// TIA Portal V17 export
// export: Created 2025-03-13T10:31:02.7493428Z, ExportSetting WithDefaults, DisplayName Totally Integrated Automation Portal, DisplayVersion V17 Update 8, DisplayName TIA Portal Openness, DisplayVersion V17 Update 8, DisplayName TIA Portal Version Control Interface, DisplayVersion V17, DisplayName SINAMICS Startdrive Advanced, DisplayVersion V17 SP2, DisplayName SINAMICS Startdrive G110M, G120, G120C, G120D, G120P, G115D, DisplayVersion V17 SP2, DisplayName SINAMICS Startdrive G130, G150, S120, S150, SINAMICS MV, S210, DisplayVersion V17 SP2, DisplayName STEP 7 Professional, DisplayVersion V17 Update 8, DisplayName SINUMERIK ONE STEP 7 Toolbox, DisplayVersion V17 Update 12, DisplayName SINUMERIK 840D sl STEP 7 Toolbox, DisplayVersion V17 Update 12, DisplayName STEP 7 Safety, DisplayVersion V17 Update 6, DisplayName WinCC Advanced, DisplayVersion V17 Update 8
DATA_BLOCK "DB1030_TEST_STOP"   // DB1030
{ S7_Optimized_Access := 'FALSE'; DB_Accessible_From_OPC_UA := 'FALSE' }
AUTHOR : ETXETAR
VERSION : 1.0
// stored: AutoNumber false, DBAccessibleFromOPCUA false, DBAccessibleFromWebserver true, IsOnlyStoredInLoadMemory false, IsWriteProtectedInAS false
   VAR
      TEST_STP_GEN_COND : Bool;   // TEST STOP GENERAL CONDITIONS / GENERAL CONDITIONS
      TEST_STP_INIT_COND : Bool;   // TEST STOP INITIAL CONDITIONS / INITIAL CONDITIONS
      TST_STP_FIRST_SCAN_REQUEST : Bool;   // FIRST SCAN REQUEST
      TEST_STP_START_REQ : Bool;   // TEST STOP START REQUEST / START REQUEST
      TEST_STP_CMD : Bool;   // TEST STOP COMMAND / COMMAND
      TEST_STP_CMD_P : Bool;   // TEST STOP COMMAND PULSE / COMMAND PULSE
      TEST_STP_SQ_IN_PROCESS : Bool;   // TEST STOP SEQUENCE IN PROCESS / SEQUENCE IN PROCESS
      TEST_STP_TST_BRK_AX_1 : Bool;   // TEST STOP TEST BRAKE AXIS 1 / BRAKE TEST AXIS 1
      TEST_STP_TST_BRK_AX_2 : Bool;   // TEST STOP TEST BRAKE AXIS 2 / BRAKE TEST AXIS 2
      TEST_STP_TST_BRK_AX_3 : Bool;   // TEST STOP TEST BRAKE AXIS 3 / BRAKE TEST AXIS 3
      TEST_STP_TST_BRK_AX_4 : Bool;   // TEST STOP TEST BRAKE AXIS 4 / BRAKE TEST AXIS 4
      TEST_STP_TST_BRK_AX_5 : Bool;   // TEST STOP TEST BRAKE AXIS 5 / BRAKE TEST AXIS 5
      TEST_STP_TST_BRK_AX_6 : Bool;   // TEST STOP TEST BRAKE AXIS 6 / BRAKE TEST AXIS 6
      TEST_STP_TST_BRK_AX_7 : Bool;   // TEST STOP TEST BRAKE AXIS 7 / BRAKE TEST AXIS 7
      TEST_STP_TST_BRK_AX_8 : Bool;   // TEST STOP TEST BRAKE AXIS 8 / BRAKE TEST AXIS 8
      TEST_STP_TST_BRK_AX_9 : Bool;   // TEST STOP TEST BRAKE AXIS 9 / BRAKE TEST AXIS 9
      TEST_STP_TST_BRK_AX_10 : Bool;   // TEST STOP TEST BRAKE AXIS 10 / BRAKE TEST AXIS 10
      TEST_STP_TST_BRK_AX_11 : Bool;   // TEST STOP TEST BRAKE AXIS 11 / BRAKE TEST AXIS 11
      TEST_STP_TST_BRK_AX_12 : Bool;   // TEST STOP TEST BRAKE AXIS 12 / BRAKE TEST AXIS 12
      TEST_STP_TST_BRK_AX_13 : Bool;   // TEST STOP TEST BRAKE AXIS 13 / BRAKE TEST AXIS 13
      TEST_STP_TST_BRK_AX_14 : Bool;   // TEST STOP TEST BRAKE AXIS 14 / BRAKE TEST AXIS 14
      TEST_STP_TST_BRK_AX_15 : Bool;   // TEST STOP TEST BRAKE AXIS15 / BRAKE TEST AXIS 15
      TEST_STP_TST_BRK_AX_16 : Bool;   // TEST STOP TEST BRAKE AXIS 16 / BRAKE TEST AXIS 16
      TEST_STP_TST_BRK_AX_17 : Bool;   // TEST STOP TEST BRAKE AXIS 17 / BRAKE TEST AXIS 17
      TEST_STP_TST_BRK_AX_18 : Bool;   // TEST STOP TEST BRAKE AXIS 18 / BRAKE TEST AXIS 18
      TEST_STP_TST_BRK_AX_19 : Bool;   // TEST STOP TEST BRAKE AXIS 19 / BRAKE TEST AXIS 19
      TEST_STP_TST_BRK_AX_20 : Bool;   // TEST STOP TEST BRAKE AXIS 20 / BRAKE TEST AXIS 20
      TEST_STP_TST_BRK_AX_21 : Bool;   // TEST STOP TEST BRAKE AXIS 21 / BRAKE TEST AXIS 21
      TEST_STP_TST_BRK_AX_22 : Bool;   // TEST STOP TEST BRAKE AXIS 22 / BRAKE TEST AXIS 22
      TEST_STP_TST_BRK_AX_23 : Bool;   // TEST STOP TEST BRAKE AXIS 23 / BRAKE TEST AXIS 23
      TEST_STP_TST_BRK_AX_24 : Bool;   // TEST STOP TEST BRAKE AXIS 24 / BRAKE TEST AXIS 24
      TEST_STP_TST_BRK_AX_25 : Bool;   // TEST STOP TEST BRAKE AXIS 25 / BRAKE TEST AXIS 25
      TEST_STP_TST_BRK_AX_26 : Bool;   // TEST STOP TEST BRAKE AXIS 26 / BRAKE TEST AXIS 26
      TEST_STP_TST_BRK_AX_27 : Bool;   // TEST STOP TEST BRAKE AXIS 27 / BRAKE TEST AXIS 27
      TEST_STP_TST_BRK_AX_28 : Bool;   // TEST STOP TEST BRAKE AXIS 28 / BRAKE TEST AXIS 28
      TEST_STP_TST_BRK_AX_29 : Bool;   // TEST STOP TEST BRAKE AXIS 29 / BRAKE TEST AXIS 29
      TEST_STP_TST_BRK_AX_30 : Bool;   // TEST STOP TEST BRAKE AXIS 30 / BRAKE TEST AXIS 30
      TEST_STP_TST_BRK_AX_31 : Bool;   // TEST STOP TEST BRAKE AXIS 31 / BRAKE TEST AXIS 31
      TEST_STP_TST_BRK_AX_32 : Bool;   // TEST STOP TEST BRAKE AXIS 32 / BRAKE TEST AXIS 32
      TEST_STP_TST_BRK_AX_33 : Bool;   // TEST STOP TEST BRAKE AXIS 33 / BRAKE TEST AXIS 33
      TEST_STP_TST_BRK_AX_34 : Bool;   // TEST STOP TEST BRAKE AXIS 34 / BRAKE TEST AXIS 34
      TEST_STP_TST_BRK_AX_35 : Bool;   // TEST STOP TEST BRAKE AXIS 35 / BRAKE TEST AXIS 35
      TEST_STP_TST_BRK_AX_36 : Bool;   // TEST STOP TEST BRAKE AXIS 36 / BRAKE TEST AXIS 36
      TEST_STP_TST_BRK_AX_37 : Bool;   // TEST STOP TEST BRAKE AXIS 37 / BRAKE TEST AXIS 37
      TEST_STP_TST_BRK_AX_38 : Bool;   // TEST STOP TEST BRAKE AXIS 38 / BRAKE TEST AXIS 38
      TEST_STP_TST_BRK_DONE : Bool;   // TEST STOP TEST BRAKE AXIS 39 / BRAKE TEST DONE
      TEST_STP_INT_P_REQ : Bool;   // TEST STOP START INTERNAL PULSES REQUEST / INTERNAL PULSES REQUEST
      TEST_STP_INT_P_REQ_AUX : Bool;   // TEST STOP START INTERNAL PULSES REQUEST PULSE / INTERNAL PULSES REQUEST AUXILIARY
      TEST_STP_INT_P_DONE : Bool;   // TEST STOP START INTERNAL PULSES DONE / INTERNAL PULSES DONE
      TEST_STP_INT_P_ANY_AX_REQ : Bool;   // TEST STOP START INTERNAL PULSES ANY AXIS REQUEST / INTERNAL PULSES ANY AXIS REQUEST
      TEST_STP_RST_PLC_CNC_SEQ : Bool;   // TEST STOP RESET PLC AND CNC / RESET PLC CNC SEQUENCE
      TEST_STP_DONE_LOCKED : Bool;   // TEST STOP DONE LOCKED / DONE LOCKED
      TEST_STP_8_HOURS : Bool;   // TEST STOP DONE LOCKED / 8 HOURS
      TEST_STP_SQ_DONE : Bool;   // TEST STOP SEQUENCE DONE / SEQUENCE DONE
      TEST_STP_SQ_TIME_EXCEEDED : Bool;   // TEST STOP SEQUENCE TIME EXCEEDED / SEQUENCE TIME EXCEEDED
      TEST_STP_FDBCK_OVERTIME : Bool;   // TEST STOP FEEDBACK TIME EXCEEDED / FEEDBACK OVERTIME
      TEST_STP_INTERNAL_P_F_AX_1 : Bool;   // TEST STOP START INTERNAL PULSES FAULT AXIS 1 / INTERNAL PULSES FAULT AXIS 1
      TEST_STP_INTERNAL_P_F_AX_2 : Bool;   // TEST STOP START INTERNAL PULSES FAULT AXIS 2 / INTERNAL PULSES FAULT AXIS 2
      TEST_STP_INTERNAL_P_F_AX_3 : Bool;   // TEST STOP START INTERNAL PULSES FAULT AXIS 3 / INTERNAL PULSES FAULT AXIS 3
      TEST_STP_INTERNAL_P_F_AX_4 : Bool;   // TEST STOP START INTERNAL PULSES FAULT AXIS 4 / INTERNAL PULSES FAULT AXIS 4
      TEST_STP_INTERNAL_P_F_AX_5 : Bool;   // TEST STOP START INTERNAL PULSES FAULT AXIS 5 / INTERNAL PULSES FAULT AXIS 5
      TEST_STP_INTERNAL_P_F_AX_6 : Bool;   // TEST STOP START INTERNAL PULSES FAULT AXIS 6 / INTERNAL PULSES FAULT AXIS 6
      TEST_STP_INTERNAL_P_F_AX_7 : Bool;   // TEST STOP START INTERNAL PULSES FAULT AXIS 7 / INTERNAL PULSES FAULT AXIS 7
      TEST_STP_INTERNAL_P_F_AX_8 : Bool;   // TEST STOP START INTERNAL PULSES FAULT AXIS 8 / INTERNAL PULSES FAULT AXIS 8
      TEST_STP_INTERNAL_P_F_AX_9 : Bool;   // TEST STOP START INTERNAL PULSES FAULT AXIS 9 / INTERNAL PULSES FAULT AXIS 9
      TEST_STP_INTERNAL_P_F_AX_10 : Bool;   // TEST STOP START INTERNAL PULSES FAULT AXIS 10 / INTERNAL PULSES FAULT AXIS 10
      TEST_STP_INTERNAL_P_F_AX_11 : Bool;   // TEST STOP START INTERNAL PULSES FAULT AXIS 11 / INTERNAL PULSES FAULT AXIS 11
      TEST_STP_INTERNAL_P_F_AX_12 : Bool;   // TEST STOP START INTERNAL PULSES FAULT AXIS 12 / INTERNAL PULSES FAULT AXIS 12
      TEST_STP_INTERNAL_P_F_AX_13 : Bool;   // TEST STOP START INTERNAL PULSES FAULT AXIS 13 / INTERNAL PULSES FAULT AXIS 13
      TEST_STP_INTERNAL_P_F_AX_14 : Bool;   // TEST STOP START INTERNAL PULSES FAULT AXIS 14 / INTERNAL PULSES FAULT AXIS 14
      TEST_STP_INTERNAL_P_F_AX_15 : Bool;   // TEST STOP START INTERNAL PULSES FAULT AXIS 15 / INTERNAL PULSES FAULT AXIS 15
      TEST_STP_INTERNAL_P_F_AX_16 : Bool;   // TEST STOP START INTERNAL PULSES FAULT AXIS 16 / INTERNAL PULSES FAULT AXIS 16
      TEST_STP_INTERNAL_P_F_AX_17 : Bool;   // TEST STOP START INTERNAL PULSES FAULT AXIS 17 / INTERNAL PULSES FAULT AXIS 17
      TEST_STP_INTERNAL_P_F_AX_18 : Bool;   // TEST STOP START INTERNAL PULSES FAULT AXIS 18 / INTERNAL PULSES FAULT AXIS 18
      TEST_STP_INTERNAL_P_F_AX_19 : Bool;   // TEST STOP START INTERNAL PULSES FAULT AXIS 19 / INTERNAL PULSES FAULT AXIS 19
      TEST_STP_INTERNAL_P_F_AX_20 : Bool;   // TEST STOP START INTERNAL PULSES FAULT AXIS 20 / INTERNAL PULSES FAULT AXIS 20
      TEST_STP_INTERNAL_P_F_AX_21 : Bool;   // TEST STOP START INTERNAL PULSES FAULT AXIS 21 / INTERNAL PULSES FAULT AXIS 21
      TEST_STP_INTERNAL_P_F_AX_22 : Bool;   // TEST STOP START INTERNAL PULSES FAULT AXIS 22 / INTERNAL PULSES FAULT AXIS 22
      TEST_STP_INTERNAL_P_F_AX_23 : Bool;   // TEST STOP START INTERNAL PULSES FAULT AXIS 23 / INTERNAL PULSES FAULT AXIS 23
      TEST_STP_INTERNAL_P_F_AX_24 : Bool;   // TEST STOP START INTERNAL PULSES FAULT AXIS 24 / INTERNAL PULSES FAULT AXIS 24
      TEST_STP_INTERNAL_P_F_AX_25 : Bool;   // TEST STOP START INTERNAL PULSES FAULT AXIS 25 / INTERNAL PULSES FAULT AXIS 25
      TEST_STP_INTERNAL_P_F_AX_26 : Bool;   // TEST STOP START INTERNAL PULSES FAULT AXIS 26 / INTERNAL PULSES FAULT AXIS 26
      TEST_STP_INTERNAL_P_F_AX_27 : Bool;   // TEST STOP START INTERNAL PULSES FAULT AXIS 27 / INTERNAL PULSES FAULT AXIS 27
      TEST_STP_INTERNAL_P_F_AX_28 : Bool;   // TEST STOP START INTERNAL PULSES FAULT AXIS 28 / INTERNAL PULSES FAULT AXIS 28
      TEST_STP_INTERNAL_P_F_AX_29 : Bool;   // TEST STOP START INTERNAL PULSES FAULT AXIS 29 / INTERNAL PULSES FAULT AXIS 29
      TEST_STP_INTERNAL_P_F_AX_30 : Bool;   // TEST STOP START INTERNAL PULSES FAULT AXIS 30 / INTERNAL PULSES FAULT AXIS 30
      TEST_STP_INTERNAL_P_F_AX_31 : Bool;   // TEST STOP START INTERNAL PULSES FAULT AXIS 31 / INTERNAL PULSES FAULT AXIS 31
      TEST_STP_INTERNAL_P_F_AX_32 : Bool;   // TEST STOP START INTERNAL PULSES FAULT AXIS 32 / INTERNAL PULSES FAULT AXIS 32
      TEST_STP_INTERNAL_P_F_AX_33 : Bool;   // TEST STOP START INTERNAL PULSES FAULT AXIS 33 / INTERNAL PULSES FAULT AXIS 33
      TEST_STP_INTERNAL_P_F_AX_34 : Bool;   // TEST STOP START INTERNAL PULSES FAULT AXIS 34 / INTERNAL PULSES FAULT AXIS 34
      TEST_STP_INTERNAL_P_F_AX_35 : Bool;   // TEST STOP START INTERNAL PULSES FAULT AXIS 35 / INTERNAL PULSES FAULT AXIS 35
      TEST_STP_INTERNAL_P_F_AX_36 : Bool;   // TEST STOP START INTERNAL PULSES FAULT AXIS 36 / INTERNAL PULSES FAULT AXIS 36
      TEST_STP_INTERNAL_P_F_AX_37 : Bool;   // TEST STOP START INTERNAL PULSES FAULT AXIS 37 / INTERNAL PULSES FAULT AXIS 37
      TEST_STP_INTERNAL_P_F_AX_38 : Bool;   // TEST STOP START INTERNAL PULSES FAULT AXIS 38 / INTERNAL PULSES FAULT AXIS 38
      TEST_STP_INTERNAL_P_F_AX_39 : Bool;   // TEST STOP START INTERNAL PULSES FAULT AXIS 39 / INTERNAL PULSES FAULT AXIS 39
      TEST_STP_TST_BRK_F_AX_1 : Bool;   // TEST STOP TEST BRAKE FAULT AXIS 1 / BRAKE TEST FAULT AXIS 1
      TEST_STP_TST_BRK_F_AX_2 : Bool;   // TEST STOP TEST BRAKE FAULT AXIS 2 / BRAKE TEST FAULT AXIS 2
      TEST_STP_TST_BRK_F_AX_3 : Bool;   // TEST STOP TEST BRAKE FAULT AXIS 3 / BRAKE TEST FAULT AXIS 3
      TEST_STP_TST_BRK_F_AX_4 : Bool;   // TEST STOP TEST BRAKE FAULT AXIS 4 / BRAKE TEST FAULT AXIS 4
      TEST_STP_TST_BRK_F_AX_5 : Bool;   // TEST STOP TEST BRAKE FAULT AXIS 5 / BRAKE TEST FAULT AXIS 5
      TEST_STP_TST_BRK_F_AX_6 : Bool;   // TEST STOP TEST BRAKE FAULT AXIS 6 / BRAKE TEST FAULT AXIS 6
      TEST_STP_TST_BRK_F_AX_7 : Bool;   // TEST STOP TEST BRAKE FAULT AXIS 7 / BRAKE TEST FAULT AXIS 7
      TEST_STP_TST_BRK_F_AX_8 : Bool;   // TEST STOP TEST BRAKE FAULT AXIS 8 / BRAKE TEST FAULT AXIS 8
      TEST_STP_TST_BRK_F_AX_9 : Bool;   // TEST STOP TEST BRAKE FAULT AXIS 9 / BRAKE TEST FAULT AXIS 9
      TEST_STP_TST_BRK_F_AX_10 : Bool;   // TEST STOP TEST BRAKE FAULT AXIS 10 / BRAKE TEST FAULT AXIS 10
      TEST_STP_TST_BRK_F_AX_11 : Bool;   // TEST STOP TEST BRAKE FAULT AXIS 11 / BRAKE TEST FAULT AXIS 11
      TEST_STP_TST_BRK_F_AX_12 : Bool;   // TEST STOP TEST BRAKE FAULT AXIS 12 / BRAKE TEST FAULT AXIS 12
      TEST_STP_TST_BRK_F_AX_13 : Bool;   // TEST STOP TEST BRAKE FAULT AXIS 13 / BRAKE TEST FAULT AXIS 13
      TEST_STP_TST_BRK_F_AX_14 : Bool;   // TEST STOP TEST BRAKE FAULT AXIS 14 / BRAKE TEST FAULT AXIS 14
      TEST_STP_TST_BRK_F_AX_15 : Bool;   // TEST STOP TEST BRAKE FAULT AXIS 15 / BRAKE TEST FAULT AXIS 15
      TEST_STP_TST_BRK_F_AX_16 : Bool;   // TEST STOP TEST BRAKE FAULT AXIS 16 / BRAKE TEST FAULT AXIS 16
      TEST_STP_TST_BRK_F_AX_17 : Bool;   // TEST STOP TEST BRAKE FAULT AXIS 17 / BRAKE TEST FAULT AXIS 17
      TEST_STP_TST_BRK_F_AX_18 : Bool;   // TEST STOP TEST BRAKE FAULT AXIS 18 / BRAKE TEST FAULT AXIS 18
      TEST_STP_TST_BRK_F_AX_19 : Bool;   // TEST STOP TEST BRAKE FAULT AXIS 19 / BRAKE TEST FAULT AXIS 19
      TEST_STP_TST_BRK_F_AX_20 : Bool;   // TEST STOP TEST BRAKE FAULT AXIS 20 / BRAKE TEST FAULT AXIS 20
      TEST_STP_TST_BRK_F_AX_21 : Bool;   // TEST STOP TEST BRAKE FAULT AXIS 21 / BRAKE TEST FAULT AXIS 21
      TEST_STP_TST_BRK_F_AX_22 : Bool;   // TEST STOP TEST BRAKE FAULT AXIS 22 / BRAKE TEST FAULT AXIS 22
      TEST_STP_TST_BRK_F_AX_23 : Bool;   // TEST STOP TEST BRAKE FAULT AXIS 23 / BRAKE TEST FAULT AXIS 23
      TEST_STP_TST_BRK_F_AX_24 : Bool;   // TEST STOP TEST BRAKE FAULT AXIS 24 / BRAKE TEST FAULT AXIS 24
      TEST_STP_TST_BRK_F_AX_25 : Bool;   // TEST STOP TEST BRAKE FAULT AXIS 25 / BRAKE TEST FAULT AXIS 25
      TEST_STP_TST_BRK_F_AX_26 : Bool;   // TEST STOP TEST BRAKE FAULT AXIS 26 / BRAKE TEST FAULT AXIS 26
      TEST_STP_TST_BRK_F_AX_27 : Bool;   // TEST STOP TEST BRAKE FAULT AXIS 27 / BRAKE TEST FAULT AXIS 27
      TEST_STP_TST_BRK_F_AX_28 : Bool;   // TEST STOP TEST BRAKE FAULT AXIS 28 / BRAKE TEST FAULT AXIS 28
      TEST_STP_TST_BRK_F_AX_29 : Bool;   // TEST STOP TEST BRAKE FAULT AXIS 29 / BRAKE TEST FAULT AXIS 29
      TEST_STP_TST_BRK_F_AX_30 : Bool;   // TEST STOP TEST BRAKE FAULT AXIS 30 / BRAKE TEST FAULT AXIS 30
      TEST_STP_TST_BRK_F_AX_31 : Bool;   // TEST STOP TEST BRAKE FAULT AXIS 31 / BRAKE TEST FAULT AXIS 31
      TEST_STP_TST_BRK_F_AX_32 : Bool;   // TEST STOP TEST BRAKE FAULT AXIS 32 / BRAKE TEST FAULT AXIS 32
      TEST_STP_TST_BRK_F_AX_33 : Bool;   // TEST STOP TEST BRAKE FAULT AXIS 33 / BRAKE TEST FAULT AXIS 33
      TEST_STP_TST_BRK_F_AX_34 : Bool;   // TEST STOP TEST BRAKE FAULT AXIS 34 / BRAKE TEST FAULT AXIS 34
      TEST_STP_TST_BRK_F_AX_35 : Bool;   // TEST STOP TEST BRAKE FAULT AXIS 35 / BRAKE TEST FAULT AXIS 35
      TEST_STP_TST_BRK_F_AX_36 : Bool;   // TEST STOP TEST BRAKE FAULT AXIS 36 / BRAKE TEST FAULT AXIS 36
      TEST_STP_TST_BRK_F_AX_37 : Bool;   // TEST STOP TEST BRAKE FAULT AXIS 37 / BRAKE TEST FAULT AXIS 37
      TEST_STP_TST_BRK_F_AX_38 : Bool;   // TEST STOP TEST BRAKE FAULT AXIS 38 / BRAKE TEST FAULT AXIS 38
      TEST_STP_TST_BRK_F_AX_39 : Bool;   // TEST STOP TEST BRAKE FAULT AXIS 39 / BRAKE TEST FAULT AXIS 39
      TEST_STP_START_GC_H : Bool;   // START TEST STOP GENERAL CONDITIONS HELP / START GENERAL CONDITIONS HELP
      TEST_STP_START_IC_H : Bool;   // START TEST STOP INITIAL CONDITIONS HELP / START INITIAL CONDITIONS HELP
      TEST_STP_STOP_GC_H : Bool;   // STOP TEST STOP GENERAL CONDITIONS HELP / STOP GENERAL CONDITIONS HELP
      TEST_STP_STOP_IC_H : Bool;   // STOP TEST STOP INITIAL CONDITIONS HELP / STOP INITIAL CONDITIONS HELP
      IS_ALARMS : Bool;   // IMMEDIATE STOP ALARMS
      TIMER_TEST_STP_INT_P_REQ_AUX { S7_SetPoint := 'True'} : TON_TIME;   // INTERNAL PULSES REQUEST AUXILIARY TIMER
      TIMER_TEST_STP_8H_AUTO_REQ { S7_SetPoint := 'True'} : TON_TIME;   // 8H AUTO REQUEST TIMER
      TIMER_TEST_STP_TIME_EXCEEDED { S7_SetPoint := 'True'} : TON_TIME;   // TIME EXCEEDED TIMER
   END_VAR
BEGIN
   TIMER_TEST_STP_INT_P_REQ_AUX.PT := T#1s;
   TIMER_TEST_STP_8H_AUTO_REQ.PT := T#8H;
   TIMER_TEST_STP_TIME_EXCEEDED.PT := T#40s;
END_DATA_BLOCK
